// TIA Portal project "sorting colo by robot arm" (V15)
// Vorlageprojekt für das Buch mit Zielsystem S7-1200

(* hardware
DEVICE "S7-1200-Station_1"  S7-1200 Station
   slot 0: "Baugruppenträger_0"  Rack  V1.0
   slot 1: "PLC_1"  CPU 1211C DC/DC/DC  6ES7 211-1AE40-0XB0  V4.1
*)

// ===== PLC "PLC_1"  CPU 1211C DC/DC/DC =====

VAR_GLOBAL   // PLC tag table "Standard-Variablentabelle"
   "START" AT %I0.0 : Bool;
   "STOP" AT %I0.1 : Bool;
   "BLUE SENSOR" AT %I0.2 : Bool;
   "GREEN SENSOR" AT %I0.3 : Bool;
   "SENSOR 1" AT %I0.4 : Bool;
   "SENSOR 2" AT %I0.5 : Bool;
   "SENSOR 3" AT %I0.6 : Bool;
   "SENSOR 4" AT %I0.7 : Bool;
   "DETECT 1" AT %I1.0 : Bool;
   "DETECT 2" AT %I1.1 : Bool;
   "MOVING X 1" AT %I1.2 : Bool;
   "MOVING X2" AT %I1.3 : Bool;
   "MOVING Z1" AT %I1.4 : Bool;
   "MOVING Z2" AT %I1.5 : Bool;
   "BELT 6M 1" AT %Q0.0 : Bool;
   "BELT 6M 3" AT %Q0.2 : Bool;
   "BELT 4M 1" AT %Q0.3 : Bool;
   "BELT 4M 2" AT %Q0.4 : Bool;
   "WHEEL" AT %Q0.5 : Bool;
   "WHEEL RIGHT" AT %Q0.6 : Bool;
   "WHEEL LEFT" AT %Q0.7 : Bool;
   "MOVE X1" AT %Q1.0 : Bool;
   "MOVE X2" AT %Q1.1 : Bool;
   "MOVE Z1" AT %Q1.2 : Bool;
   "MOVE Z2" AT %Q1.3 : Bool;
   "GRAB 1" AT %Q1.4 : Bool;
   "GRAB 2" AT %Q1.5 : Bool;
   "BELT 6M 2" AT %Q0.1 : Bool;
   "X" AT %M0.0 : Bool;   // X
   "Tag_1" AT %M7.0 : Bool;
   "Tag_2" AT %M7.1 : Bool;
   "M2 move z1" AT %M0.1 : Bool;
   "M1 move z1" AT %M0.2 : Bool;
   "Tag_3" AT %M7.3 : Bool;
   "Tag_4" AT %M7.4 : Bool;
   "Tag_5" AT %M7.5 : Bool;
   "Tag_6" AT %M7.6 : Bool;
   "Tag_7" AT %M7.7 : Bool;
   "Tag_8" AT %M8.0 : Bool;
   "Tag_9" AT %M8.1 : Bool;
   "Tag_10" AT %M8.2 : Bool;
   "Tag_11" AT %M8.3 : Bool;
   "Tag_12" AT %M8.4 : Bool;
   "Tag_13" AT %M8.5 : Bool;
   "Tag_14" AT %M5.0 : Bool;
   "M1 moving Z2" AT %M5.1 : Bool;
   "Tag_15" AT %M5.3 : Bool;
   "Tag_16" AT %M5.4 : Bool;
   "Tag_17" AT %M5.6 : Bool;
   "Tag_18" AT %M5.5 : Bool;
   "M2 move Z2" AT %M5.2 : Bool;
   "Tag_19" AT %M5.7 : Bool;
   "Tag_20" AT %M6.0 : Bool;
   "Tag_21" AT %QD16 : DWord;
   "Tag_22" AT %QD20 : DWord;
END_VAR

// folder: System blocks/Program resources

DATA_BLOCK "c1"   // DB1
{ S7_Optimized_Access := 'TRUE' }
AUTHOR : Simatic
FAMILY : IEC
NAME : CNTR
VERSION : 1.0
// stored: InstanceOfName IEC_COUNTER
"IEC_COUNTER"
BEGIN
END_DATA_BLOCK

DATA_BLOCK "c2"   // DB2
{ S7_Optimized_Access := 'TRUE' }
AUTHOR : Simatic
FAMILY : IEC
NAME : CNTR
VERSION : 1.0
// stored: InstanceOfName IEC_COUNTER
"IEC_COUNTER"
BEGIN
END_DATA_BLOCK

// folder: (top level)

FUNCTION "MHJ-PLC-Lab-Function-S71200" : Void   // FC9000, SCL
{ S7_Optimized_Access := 'TRUE' }
VERSION : 0.1
   VAR_TEMP
      rdTimeReturn : Int;
      outputTime : DTL;
      SyncVal : Byte;
      forVal : Int;
      forVal_2 : Int;
      Value : Byte;
   END_VAR
   VAR CONSTANT
      CompVal : Byte := 16#34;
      Value_01 : Byte := 16#11;
      Value_01_DW : DWord := 16#A165_D992;
      Value_02_DW : DWord := 16#58BE_4401;
   END_VAR
BEGIN

   #Value:=PEEK(area := 16#82,
        dbNumber := 0,
        byteOffset := 511);
   #Value := #Value + 1;

   POKE(area := 16#82,
        dbNumber := 0,
        byteOffset := 511,
        value := #Value);

   POKE(area:=16#81,
        dbNumber:=0,
        byteOffset:=1016,
        value:=#Value_01_DW);
   POKE(area := 16#81,
        dbNumber := 0,
        byteOffset := 1020,
        value := #Value_02_DW);

   POKE(area := 16#81,
        dbNumber := 0,
        byteOffset := 511,
        value := B#16#00);

   FOR #forVal := 0 TO 120 DO
       FOR #forVal_2:=0 TO 10 DO
           #rdTimeReturn:=RD_SYS_T(#outputTime);
           #rdTimeReturn := WR_SYS_T(#outputTime);
           #rdTimeReturn := RD_SYS_T(#outputTime);
           #rdTimeReturn := WR_SYS_T(#outputTime);
       END_FOR;
       #SyncVal:= PEEK(area := 16#81,
                      dbNumber := 0,
                      byteOffset := 511);
       IF #SyncVal = #CompVal THEN
          GOTO M_1;
       END_IF;
   END_FOR;
   RETURN;

   M_1:
   POKE(area := 16#81,
        dbNumber := 0,
        byteOffset := 511,
        value := B#16#0);
END_FUNCTION

ORGANIZATION_BLOCK "Main"   // OB1, LAD, ProgramCycle
TITLE = "Main Program Sweep (Cycle)"
{ S7_Optimized_Access := 'TRUE' }
VERSION : 0.1
   VAR_INPUT
      Initial_Call : Bool;   // Initial call of this OB
      Remanence : Bool;   // =True, if remanent data are available
   END_VAR
   VAR_TEMP   // added for the SCL form of the ladder/FBD networks
      _w1 : Bool;
      _w2 : Bool;
      _w3 : Bool;
      _w4 : Bool;
   END_VAR
BEGIN

REGION Network 1: Konnektierungsbaustein für PLC-Lab
   // Im Netzwerk 1 wird der Konnektierungsbaustein für PLC-Lab aufgerufen.
   // Dieser Aufruf darf nicht entfernt werden!
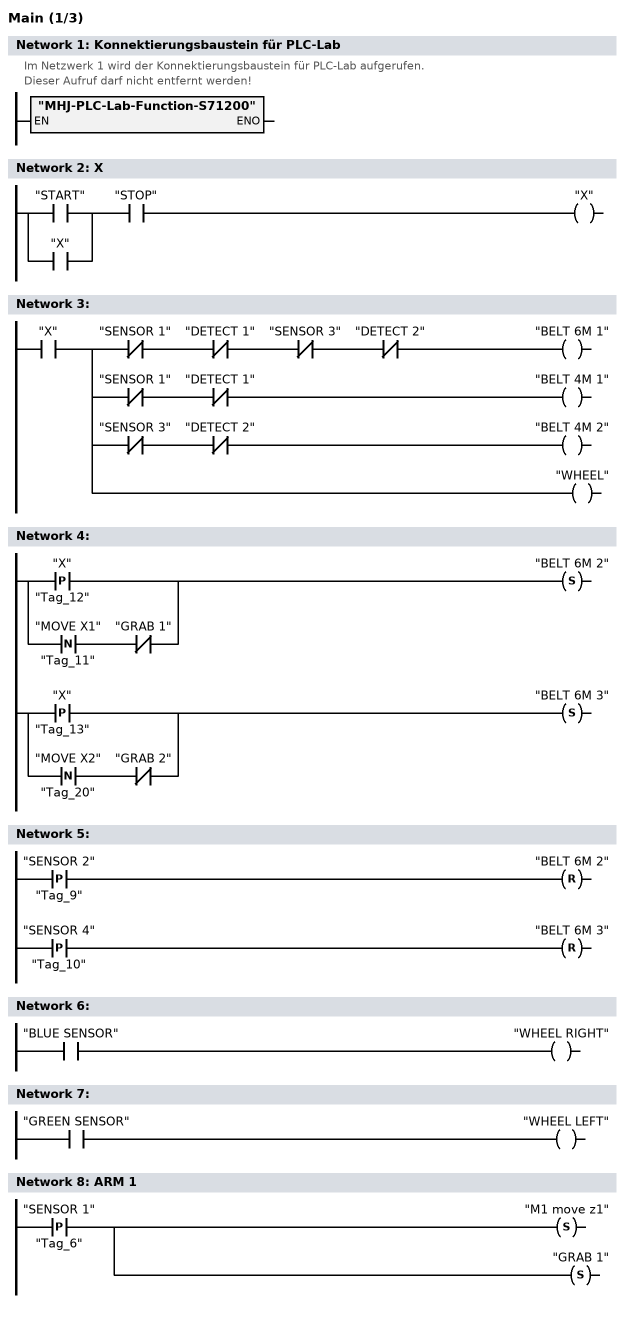
   RUNG wire#powerrail
      "MHJ-PLC-Lab-Function-S71200"()
   END_RUNG
   // the same network as SCL:
   "MHJ-PLC-Lab-Function-S71200"();
END_REGION

REGION Network 2: X
   RUNG wire#powerrail
      Contact( "START" )
      wire#w1
      Contact( "STOP" )
      Coil( "X" )
   END_RUNG
   RUNG wire#powerrail
      Contact( "X" )
   END_RUNG wire#w1
   // the same network as SCL:
   "X" := ("START" OR "X") AND "STOP";
END_REGION

REGION Network 3
   RUNG wire#powerrail
      Contact( "X" )
      wire#w1
      I_Contact( "SENSOR 1" )
      I_Contact( "DETECT 1" )
      I_Contact( "SENSOR 3" )
      I_Contact( "DETECT 2" )
      Coil( "BELT 6M 1" )
   END_RUNG
   RUNG wire#w1
      I_Contact( "SENSOR 1" )
      I_Contact( "DETECT 1" )
      Coil( "BELT 4M 1" )
   END_RUNG
   RUNG wire#w1
      I_Contact( "SENSOR 3" )
      I_Contact( "DETECT 2" )
      Coil( "BELT 4M 2" )
   END_RUNG
   RUNG wire#w1
      Coil( "WHEEL" )
   END_RUNG
   // the same network as SCL:
   "BELT 6M 1" := "X" AND NOT "SENSOR 1" AND NOT "DETECT 1" AND NOT "SENSOR 3" AND NOT "DETECT 2";
   "BELT 4M 1" := "X" AND NOT "SENSOR 1" AND NOT "DETECT 1";
   "BELT 4M 2" := "X" AND NOT "SENSOR 3" AND NOT "DETECT 2";
   "WHEEL" := "X";
END_REGION

REGION Network 4
   RUNG wire#powerrail
      P_Contact(operand := "X", bit := "Tag_12")
      wire#w1
      S_Coil( "BELT 6M 2" )
   END_RUNG
   RUNG wire#powerrail
      N_Contact(operand := "MOVE X1", bit := "Tag_11")
      I_Contact( "GRAB 1" )
   END_RUNG wire#w1
   RUNG wire#powerrail
      P_Contact(operand := "X", bit := "Tag_13")
      wire#w2
      S_Coil( "BELT 6M 3" )
   END_RUNG
   RUNG wire#powerrail
      N_Contact(operand := "MOVE X2", bit := "Tag_20")
      I_Contact( "GRAB 2" )
   END_RUNG wire#w2
   // the same network as SCL:
   #_w1 := "X" AND NOT "Tag_12";   // rising edge of "X"
   "Tag_12" := "X";
   #_w2 := NOT "MOVE X1" AND "Tag_11";   // falling edge of "MOVE X1"
   "Tag_11" := "MOVE X1";
   IF #_w1 OR (#_w2 AND NOT "GRAB 1") THEN "BELT 6M 2" := TRUE; END_IF;
   #_w3 := "X" AND NOT "Tag_13";   // rising edge of "X"
   "Tag_13" := "X";
   #_w4 := NOT "MOVE X2" AND "Tag_20";   // falling edge of "MOVE X2"
   "Tag_20" := "MOVE X2";
   IF #_w3 OR (#_w4 AND NOT "GRAB 2") THEN "BELT 6M 3" := TRUE; END_IF;
END_REGION

REGION Network 5
   RUNG wire#powerrail
      P_Contact(operand := "SENSOR 2", bit := "Tag_9")
      R_Coil( "BELT 6M 2" )
   END_RUNG
   RUNG wire#powerrail
      P_Contact(operand := "SENSOR 4", bit := "Tag_10")
      R_Coil( "BELT 6M 3" )
   END_RUNG
   // the same network as SCL:
   #_w1 := "SENSOR 2" AND NOT "Tag_9";   // rising edge of "SENSOR 2"
   "Tag_9" := "SENSOR 2";
   IF #_w1 THEN "BELT 6M 2" := FALSE; END_IF;
   #_w2 := "SENSOR 4" AND NOT "Tag_10";   // rising edge of "SENSOR 4"
   "Tag_10" := "SENSOR 4";
   IF #_w2 THEN "BELT 6M 3" := FALSE; END_IF;
END_REGION

REGION Network 6
   RUNG wire#powerrail
      Contact( "BLUE SENSOR" )
      Coil( "WHEEL RIGHT" )
   END_RUNG
   // the same network as SCL:
   "WHEEL RIGHT" := "BLUE SENSOR";
END_REGION

REGION Network 7
   RUNG wire#powerrail
      Contact( "GREEN SENSOR" )
      Coil( "WHEEL LEFT" )
   END_RUNG
   // the same network as SCL:
   "WHEEL LEFT" := "GREEN SENSOR";
END_REGION

REGION Network 8: ARM 1
   RUNG wire#powerrail
      P_Contact(operand := "SENSOR 1", bit := "Tag_6")
      wire#w1
      S_Coil( "M1 move z1" )
   END_RUNG
   RUNG wire#w1
      S_Coil( "GRAB 1" )
   END_RUNG
   // the same network as SCL:
   #_w1 := "SENSOR 1" AND NOT "Tag_6";   // rising edge of "SENSOR 1"
   "Tag_6" := "SENSOR 1";
   IF #_w1 THEN
       "M1 move z1" := TRUE;
       "GRAB 1" := TRUE;
   END_IF;
END_REGION

REGION Network 9
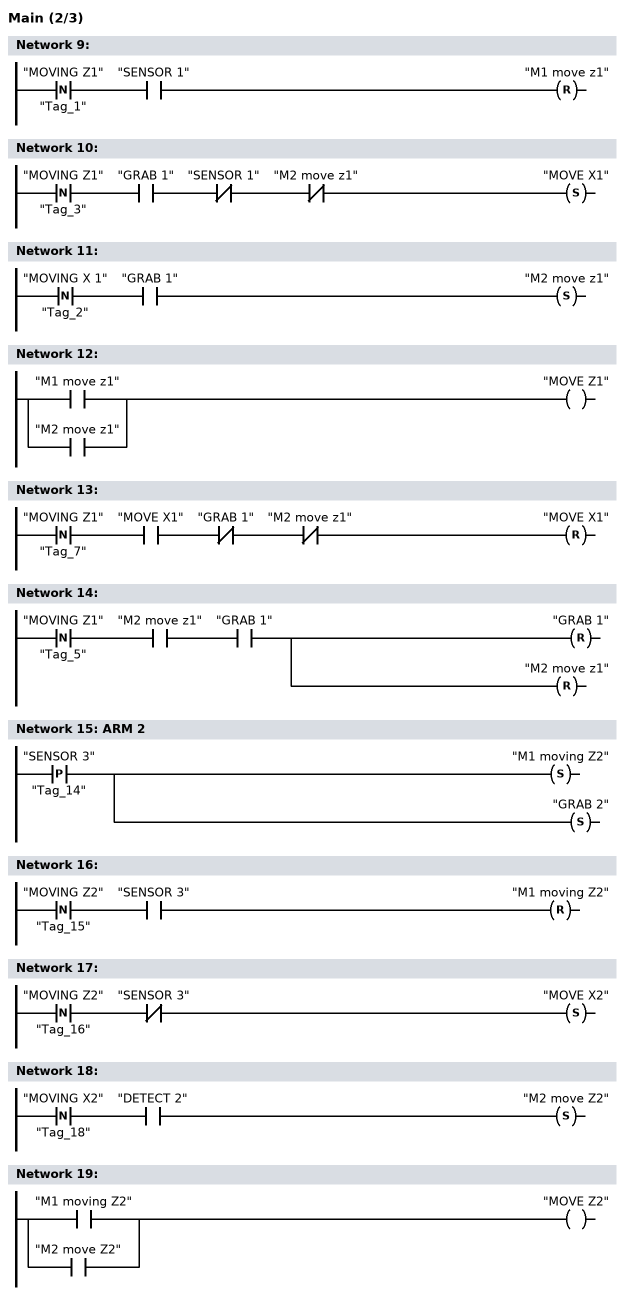
   RUNG wire#powerrail
      N_Contact(operand := "MOVING Z1", bit := "Tag_1")
      Contact( "SENSOR 1" )
      R_Coil( "M1 move z1" )
   END_RUNG
   // the same network as SCL:
   #_w1 := NOT "MOVING Z1" AND "Tag_1";   // falling edge of "MOVING Z1"
   "Tag_1" := "MOVING Z1";
   IF #_w1 AND "SENSOR 1" THEN "M1 move z1" := FALSE; END_IF;
END_REGION

REGION Network 10
   RUNG wire#powerrail
      N_Contact(operand := "MOVING Z1", bit := "Tag_3")
      Contact( "GRAB 1" )
      I_Contact( "SENSOR 1" )
      I_Contact( "M2 move z1" )
      S_Coil( "MOVE X1" )
   END_RUNG
   // the same network as SCL:
   #_w1 := NOT "MOVING Z1" AND "Tag_3";   // falling edge of "MOVING Z1"
   "Tag_3" := "MOVING Z1";
   IF #_w1 AND "GRAB 1" AND NOT "SENSOR 1" AND NOT "M2 move z1" THEN "MOVE X1" := TRUE; END_IF;
END_REGION

REGION Network 11
   RUNG wire#powerrail
      N_Contact(operand := "MOVING X 1", bit := "Tag_2")
      Contact( "GRAB 1" )
      S_Coil( "M2 move z1" )
   END_RUNG
   // the same network as SCL:
   #_w1 := NOT "MOVING X 1" AND "Tag_2";   // falling edge of "MOVING X 1"
   "Tag_2" := "MOVING X 1";
   IF #_w1 AND "GRAB 1" THEN "M2 move z1" := TRUE; END_IF;
END_REGION

REGION Network 12
   RUNG wire#powerrail
      Contact( "M1 move z1" )
      wire#w1
      Coil( "MOVE Z1" )
   END_RUNG
   RUNG wire#powerrail
      Contact( "M2 move z1" )
   END_RUNG wire#w1
   // the same network as SCL:
   "MOVE Z1" := "M1 move z1" OR "M2 move z1";
END_REGION

REGION Network 13
   RUNG wire#powerrail
      N_Contact(operand := "MOVING Z1", bit := "Tag_7")
      Contact( "MOVE X1" )
      I_Contact( "GRAB 1" )
      I_Contact( "M2 move z1" )
      R_Coil( "MOVE X1" )
   END_RUNG
   // the same network as SCL:
   #_w1 := NOT "MOVING Z1" AND "Tag_7";   // falling edge of "MOVING Z1"
   "Tag_7" := "MOVING Z1";
   IF #_w1 AND "MOVE X1" AND NOT "GRAB 1" AND NOT "M2 move z1" THEN "MOVE X1" := FALSE; END_IF;
END_REGION

REGION Network 14
   RUNG wire#powerrail
      N_Contact(operand := "MOVING Z1", bit := "Tag_5")
      Contact( "M2 move z1" )
      Contact( "GRAB 1" )
      wire#w1
      R_Coil( "GRAB 1" )
   END_RUNG
   RUNG wire#w1
      R_Coil( "M2 move z1" )
   END_RUNG
   // the same network as SCL:
   #_w1 := NOT "MOVING Z1" AND "Tag_5";   // falling edge of "MOVING Z1"
   "Tag_5" := "MOVING Z1";
   #_w2 := #_w1 AND "M2 move z1" AND "GRAB 1";
   IF #_w2 THEN
       "GRAB 1" := FALSE;
       "M2 move z1" := FALSE;
   END_IF;
END_REGION

REGION Network 15: ARM 2
   RUNG wire#powerrail
      P_Contact(operand := "SENSOR 3", bit := "Tag_14")
      wire#w1
      S_Coil( "M1 moving Z2" )
   END_RUNG
   RUNG wire#w1
      S_Coil( "GRAB 2" )
   END_RUNG
   // the same network as SCL:
   #_w1 := "SENSOR 3" AND NOT "Tag_14";   // rising edge of "SENSOR 3"
   "Tag_14" := "SENSOR 3";
   IF #_w1 THEN
       "M1 moving Z2" := TRUE;
       "GRAB 2" := TRUE;
   END_IF;
END_REGION

REGION Network 16
   RUNG wire#powerrail
      N_Contact(operand := "MOVING Z2", bit := "Tag_15")
      Contact( "SENSOR 3" )
      R_Coil( "M1 moving Z2" )
   END_RUNG
   // the same network as SCL:
   #_w1 := NOT "MOVING Z2" AND "Tag_15";   // falling edge of "MOVING Z2"
   "Tag_15" := "MOVING Z2";
   IF #_w1 AND "SENSOR 3" THEN "M1 moving Z2" := FALSE; END_IF;
END_REGION

REGION Network 17
   RUNG wire#powerrail
      N_Contact(operand := "MOVING Z2", bit := "Tag_16")
      I_Contact( "SENSOR 3" )
      S_Coil( "MOVE X2" )
   END_RUNG
   // the same network as SCL:
   #_w1 := NOT "MOVING Z2" AND "Tag_16";   // falling edge of "MOVING Z2"
   "Tag_16" := "MOVING Z2";
   IF #_w1 AND NOT "SENSOR 3" THEN "MOVE X2" := TRUE; END_IF;
END_REGION

REGION Network 18
   RUNG wire#powerrail
      N_Contact(operand := "MOVING X2", bit := "Tag_18")
      Contact( "DETECT 2" )
      S_Coil( "M2 move Z2" )
   END_RUNG
   // the same network as SCL:
   #_w1 := NOT "MOVING X2" AND "Tag_18";   // falling edge of "MOVING X2"
   "Tag_18" := "MOVING X2";
   IF #_w1 AND "DETECT 2" THEN "M2 move Z2" := TRUE; END_IF;
END_REGION

REGION Network 19
   RUNG wire#powerrail
      Contact( "M1 moving Z2" )
      wire#w1
      Coil( "MOVE Z2" )
   END_RUNG
   RUNG wire#powerrail
      Contact( "M2 move Z2" )
   END_RUNG wire#w1
   // the same network as SCL:
   "MOVE Z2" := "M1 moving Z2" OR "M2 move Z2";
END_REGION

REGION Network 20
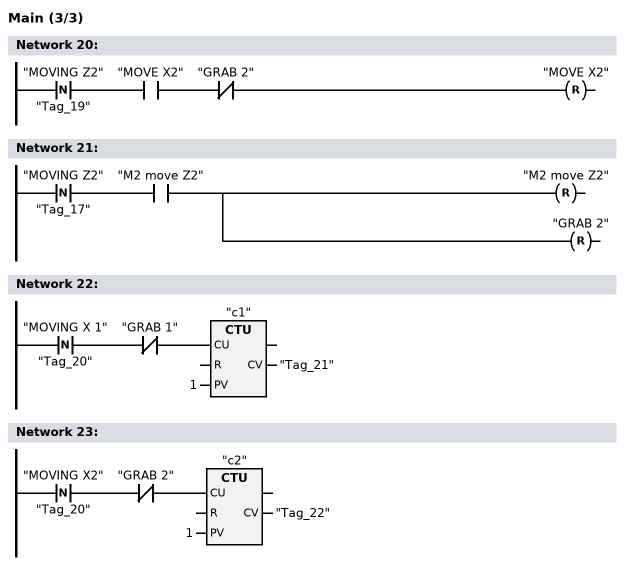
   RUNG wire#powerrail
      N_Contact(operand := "MOVING Z2", bit := "Tag_19")
      Contact( "MOVE X2" )
      I_Contact( "GRAB 2" )
      R_Coil( "MOVE X2" )
   END_RUNG
   // the same network as SCL:
   #_w1 := NOT "MOVING Z2" AND "Tag_19";   // falling edge of "MOVING Z2"
   "Tag_19" := "MOVING Z2";
   IF #_w1 AND "MOVE X2" AND NOT "GRAB 2" THEN "MOVE X2" := FALSE; END_IF;
END_REGION

REGION Network 21
   RUNG wire#powerrail
      N_Contact(operand := "MOVING Z2", bit := "Tag_17")
      Contact( "M2 move Z2" )
      wire#w1
      R_Coil( "M2 move Z2" )
   END_RUNG
   RUNG wire#w1
      R_Coil( "GRAB 2" )
   END_RUNG
   // the same network as SCL:
   #_w1 := NOT "MOVING Z2" AND "Tag_17";   // falling edge of "MOVING Z2"
   "Tag_17" := "MOVING Z2";
   #_w2 := #_w1 AND "M2 move Z2";
   IF #_w2 THEN
       "M2 move Z2" := FALSE;
       "GRAB 2" := FALSE;
   END_IF;
END_REGION

REGION Network 22
   #_w1 := NOT "MOVING X 1" AND "Tag_20";   // falling edge of "MOVING X 1"
   "Tag_20" := "MOVING X 1";
   "c1".CTU(CU := #_w1 AND NOT "GRAB 1", PV := 1, CV => "Tag_21");
END_REGION

REGION Network 23
   #_w1 := NOT "MOVING X2" AND "Tag_20";   // falling edge of "MOVING X2"
   "Tag_20" := "MOVING X2";
   "c2".CTU(CU := #_w1 AND NOT "GRAB 2", PV := 1, CV => "Tag_22");
END_REGION
END_ORGANIZATION_BLOCK